PROGRAM MAIN
VAR
	fbController		: FB_Controller();
	fbLampOnOff			: FB_LampOnOff();
	fbLampSetDirect		: FB_LampSetDirect();
	fbLampUpDown		: FB_LampUpDown();
	nSetLamp			: INT;
	bDimUp, bDimDown	: BOOL;
	bOff, bOn			: BOOL;
END_VAR

CASE nSetLamp OF
	1:
		fbController.refActiveLamp REF= fbLampOnOff;
		nSetLamp := 0;
	2:
		fbController.refActiveLamp REF= fbLampSetDirect;
		nSetLamp := 0;
	3:
		fbController.refActiveLamp REF= fbLampUpDown;
		nSetLamp := 0;
END_CASE

IF (bDimUp) THEN
	fbController.DimUp();
	bDimUp := FALSE;
END_IF

IF (bDimDown) THEN
	fbController.DimDown();
	bDimDown := FALSE;
END_IF

IF (bOff) THEN
	fbController.Off();
	bOff := FALSE;
END_IF

IF (bOn) THEN
	fbController.On();
	bOn := FALSE;
END_IF

END_PROGRAM

(* stored: Version 1.1.0.1, ProductVersion 3.1.4024.9
   POU MAIN: Id {ef33b4c1-c95d-4cf8-b9bf-7d346bd93484}, SpecialFunc None *)
